Staubli VAL3: sZone.pgx

public program sZone(tool x_tTool, point x_pPoint, frame x_fFrame, num x_Dx, num x_Dy, num x_Dz)
begin

  //in automatic mode stop immediately the robot if x_tTool is out of a box defined as:

  //x_pPoint.trsf.x + x_Dx/2 > here(x_tTool, x_fFrame).x > x_pPoint.trsf.x - x_Dx/2
  //x_pPoint.trsf.y + x_Dy/2 > here(x_tTool, x_fFrame).y > x_pPoint.trsf.y - x_Dy/2
  //x_pPoint.trsf.z + x_Dz/2 > here(x_tTool, x_fFrame).z > x_pPoint.trsf.z - x_Dz/2

  if taskStatus("sZone_"+toString("",nSzoneCount))==-1
    taskCreate "sZone_"+toString("",nSzoneCount),15,exeSzone(x_tTool,x_pPoint,x_fFrame,x_Dx,x_Dy,x_Dz)
    nSzoneCount=nSzoneCount+1
    if nSzoneCount>nMaxTask
      nSzoneCount=0
    endIf
  else
    logMsg("libSignals/sZone->can't create the task")
  endIf

end
